Fanuc KAREL source: CA0123.KL

PROGRAM CA0123
%STACKSIZE=65535
%PRIORITY=65535
%NOLOCKGROUP
VAR
G : INTEGER
I : INTEGER
R : REAL
B : BOOLEAN
S : STRING[16]
AI : ARRAY[2] OF INTEGER
AR : ARRAY[2] OF REAL
P : XYZWPR
-- UNRESOLVED DECLARATIONS (source type spelling not recovered)
-- ST : TYPE_0x1100 (type_u16=0x1100)
-- V : TYPE_0x0013 (type_u16=0x0013)
ROUTINE H1(P1 : INTEGER) : INTEGER FROM CA0123
ROUTINE H2(P1 : INTEGER) : INTEGER FROM CA0123
ROUTINE H3(P1 : INTEGER) : INTEGER FROM CA0123
ROUTINE F(P1 : INTEGER; P2 : INTEGER; P3 : INTEGER) FROM CA0123
ROUTINE H1
BEGIN
G=(G + 1)
-- UNRESOLVED_PC line 22 opcodes [2D 21 52 7F] marker_code=20
-- UNRESOLVED_PC line 23 opcodes [7F] marker_code=42
END H1
ROUTINE H2
BEGIN
G=(G + 2)
-- UNRESOLVED_PC line 27 opcodes [2D 21 52 7F] marker_code=75
-- UNRESOLVED_PC line 28 opcodes [7F] marker_code=97
END H2
ROUTINE H3
BEGIN
G=(G + 3)
-- UNRESOLVED_PC line 32 opcodes [2D 21 52 7F] marker_code=130
-- UNRESOLVED_PC line 33 opcodes [7F] marker_code=152
END H3
ROUTINE F
BEGIN
G=(G + 1)
END F
BEGIN
G=0
I=1
R=2.5
B=TRUE
S='A'
AI[1]=3
AR[1]=4.5
ST.A=5
ST.B=1087373312
-- UNSAFE_SOURCE_IR line 50: CALL_RESULT H1(ARG_1_UNRESOLVED)
-- UNSAFE_SOURCE_IR line 50: CALL_RESULT H1(ARG_1_UNRESOLVED)
-- UNSAFE_SOURCE_IR line 50: CALL_RESULT H1(ARG_1_UNRESOLVED)
-- UNSAFE_SOURCE_IR line 50: F(ARG_1_UNRESOLVED, ARG_2_UNRESOLVED, ARG_3_UNRESOLVED)
END CA0123
